// TIA Portal V20 export
// export: Created 2025-12-01T14:57:00.6413391Z, ExportSetting None, DisplayName Totally Integrated Automation Portal, DisplayVersion V20 Update 3, DisplayName TIA Portal Openness, DisplayVersion V20 Update 3, DisplayName TIA Portal Version Control Interface, DisplayVersion V20 Update 3, DisplayName STEP 7 Professional, DisplayVersion V20 Update 3, DisplayName STEP 7 Safety, DisplayVersion V20 Update 2, DisplayName WinCC Basic/Comfort/Advanced, DisplayVersion V20 Update 3, DisplayName WinCC Professional, DisplayVersion V20 Update 3, DisplayName WinCC Unified, DisplayVersion V20 Update 3
FUNCTION "FC452_TL_TR_E1E3_S2_Pres" : Void   // FC452, LAD
{ S7_Optimized_Access := 'FALSE' }
AUTHOR : TLigero
NAME : 20160208
VERSION : 3.1
// stored: AutoNumber false, SetENOAutomatically false
   VAR_INPUT
      Mesa : UInt;
      En_Tension : Bool;
      pHsMx_E1 : Bool;   // Para contar cuando se entra por E1
      pHsMx_E3 : Bool;   // Para contar cuando se entra por E3
      Termico_E1_Tx : Bool;
      Termico_S2_Tx : Bool;
      Avance_E1_Tx_Ok : Bool;
      Avance_E3_Tx_Ok : Bool;   // será el retroceso de E1
      Avance_S2_Tx_Ok : Bool;
      PosTR_E1 : Bool;
      PosTR_S2 : Bool;
      TP_E1E3_UP : Bool;
      TP_E1E3_DW : Bool;
      TP_E3E1_UP : Bool;
      TP_E3E1_DW : Bool;
      AVTF_Ent_M1 : Bool;
      AVTF_Ent_M3 : Bool;
      NXT_Avance : Bool;
      PTF_Mx_MSig : Bool;
      V_CNT_pHsMx_E1 : UDInt;
      V_CNT_pHsMx_E3 : UDInt;
      V_Paro : UDInt;
      V_CNT_ApHsMx : UDInt;
      V_TOut_Tx_Mx : UDInt;
      V_TOut_TR : UDInt;
      V_TOut_TP : UDInt;
      V_Reparto_E1_E3 : UDInt;
   END_VAR
   VAR_OUTPUT
      PTF_Ent_M1 : Bool;
      PTF_Ent_M3 : Bool;
      AVTF_Mx_MSig : Bool;
      NXT_Descarga_Act : Bool;
   END_VAR
   VAR_IN_OUT
      MemFP_Carga_E1 : Bool;
   END_VAR
   VAR_TEMP
      Mem_CNT_Aus : Bool;
      Aux_Parar : Bool;
      Mem_CNT_Pres : Bool;
      Mem_CNT_Tmp_Paro : Bool;
      TEMP_MA_TR_Pos_E1 : Bool;
      TEMP_MA_TR_Pos_S2 : Bool;
      Atasco : Bool;
      Tout_movimiento : Bool;
      tout_tope : Bool;
      ok_tension : Bool;
      V_Presencia : UDInt;
   END_VAR
   VAR_TEMP   // added for the SCL form of the ladder/FBD networks
      _w1 : Bool;
   END_VAR
BEGIN

REGION Network 1: Marca General Error
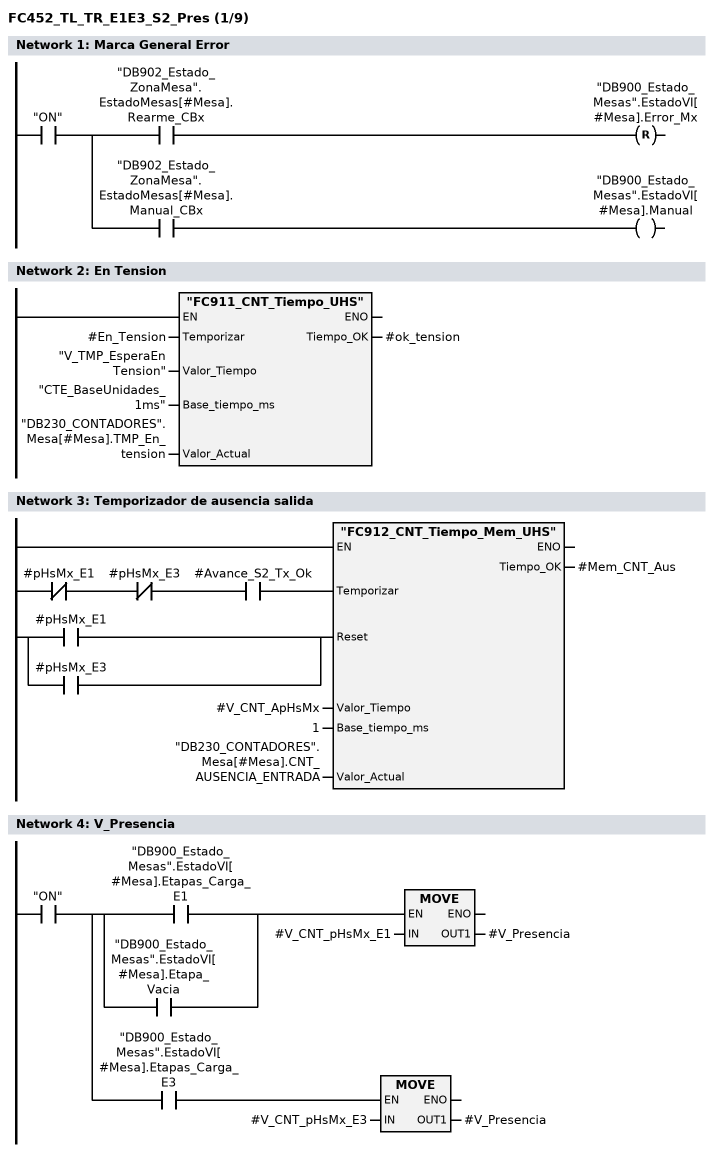
   RUNG wire#powerrail
      Contact( "ON" )
      wire#w1
      Contact( "DB902_Estado_ZonaMesa".EstadoMesas[#Mesa].Rearme_CBx )
      R_Coil( "DB900_Estado_Mesas".EstadoVI[#Mesa].Error_Mx )
   END_RUNG
   RUNG wire#w1
      Contact( "DB902_Estado_ZonaMesa".EstadoMesas[#Mesa].Manual_CBx )
      Coil( "DB900_Estado_Mesas".EstadoVI[#Mesa].Manual )
   END_RUNG
   // the same network as SCL:
   IF "ON" AND "DB902_Estado_ZonaMesa".EstadoMesas[#Mesa].Rearme_CBx THEN
       "DB900_Estado_Mesas".EstadoVI[#Mesa].Error_Mx := FALSE;
   END_IF;
   "DB900_Estado_Mesas".EstadoVI[#Mesa].Manual := "ON" AND "DB902_Estado_ZonaMesa".EstadoMesas[#Mesa].Manual_CBx;
END_REGION

REGION Network 2: En Tension
   RUNG wire#powerrail
      "FC911_CNT_Tiempo_UHS"(Temporizar := #En_Tension, Valor_Tiempo := "V_TMP_EsperaEnTension", Base_tiempo_ms := "CTE_BaseUnidades_1ms", Valor_Actual := "DB230_CONTADORES".Mesa[#Mesa].TMP_En_tension, Tiempo_OK => #ok_tension)
   END_RUNG
   // the same network as SCL:
   "FC911_CNT_Tiempo_UHS"(Temporizar := #En_Tension,
                          Valor_Tiempo := "V_TMP_EsperaEnTension",
                          Base_tiempo_ms := "CTE_BaseUnidades_1ms",
                          Valor_Actual := "DB230_CONTADORES".Mesa[#Mesa].TMP_En_tension,
                          Tiempo_OK => #ok_tension);
END_REGION

REGION Network 3: Temporizador de ausencia salida
   RUNG wire#powerrail
      "FC912_CNT_Tiempo_Mem_UHS"(Temporizar := wire#w1, Reset := wire#w2, Valor_Tiempo := #V_CNT_ApHsMx, Base_tiempo_ms := 1, Valor_Actual := "DB230_CONTADORES".Mesa[#Mesa].CNT_AUSENCIA_ENTRADA, Tiempo_OK => #Mem_CNT_Aus)
   END_RUNG
   RUNG wire#powerrail
      I_Contact( #pHsMx_E1 )
      I_Contact( #pHsMx_E3 )
      Contact( #Avance_S2_Tx_Ok )
   END_RUNG wire#w1
   RUNG wire#powerrail
      Contact( #pHsMx_E1 )
   END_RUNG wire#w2
   RUNG wire#powerrail
      Contact( #pHsMx_E3 )
   END_RUNG wire#w2
   // the same network as SCL:
   "FC912_CNT_Tiempo_Mem_UHS"(Temporizar := NOT #pHsMx_E1 AND NOT #pHsMx_E3 AND #Avance_S2_Tx_Ok,
                           Reset := #pHsMx_E1 OR #pHsMx_E3,
                           Valor_Tiempo := #V_CNT_ApHsMx,
                           Base_tiempo_ms := 1,
                           Valor_Actual := "DB230_CONTADORES".Mesa[#Mesa].CNT_AUSENCIA_ENTRADA,
                           Tiempo_OK => #Mem_CNT_Aus);
END_REGION

REGION Network 4: V_Presencia
   RUNG wire#powerrail
      Contact( "ON" )
      wire#w1
      Contact( "DB900_Estado_Mesas".EstadoVI[#Mesa].Etapas_Carga_E1 )
      wire#w2
      Move(in := #V_CNT_pHsMx_E1, out1 => #V_Presencia)
   END_RUNG
   RUNG wire#w1
      Contact( "DB900_Estado_Mesas".EstadoVI[#Mesa].Etapa_Vacia )
   END_RUNG wire#w2
   RUNG wire#w1
      Contact( "DB900_Estado_Mesas".EstadoVI[#Mesa].Etapas_Carga_E3 )
      Move(in := #V_CNT_pHsMx_E3, out1 => #V_Presencia)
   END_RUNG
   // the same network as SCL:
   IF "ON" AND ("DB900_Estado_Mesas".EstadoVI[#Mesa].Etapas_Carga_E1 OR "DB900_Estado_Mesas".EstadoVI[#Mesa].Etapa_Vacia) THEN
       #V_Presencia := #V_CNT_pHsMx_E1;
   END_IF;
   IF "ON" AND "DB900_Estado_Mesas".EstadoVI[#Mesa].Etapas_Carga_E3 THEN
       #V_Presencia := #V_CNT_pHsMx_E3;
   END_IF;
END_REGION

REGION Network 5: Temporizador presencia
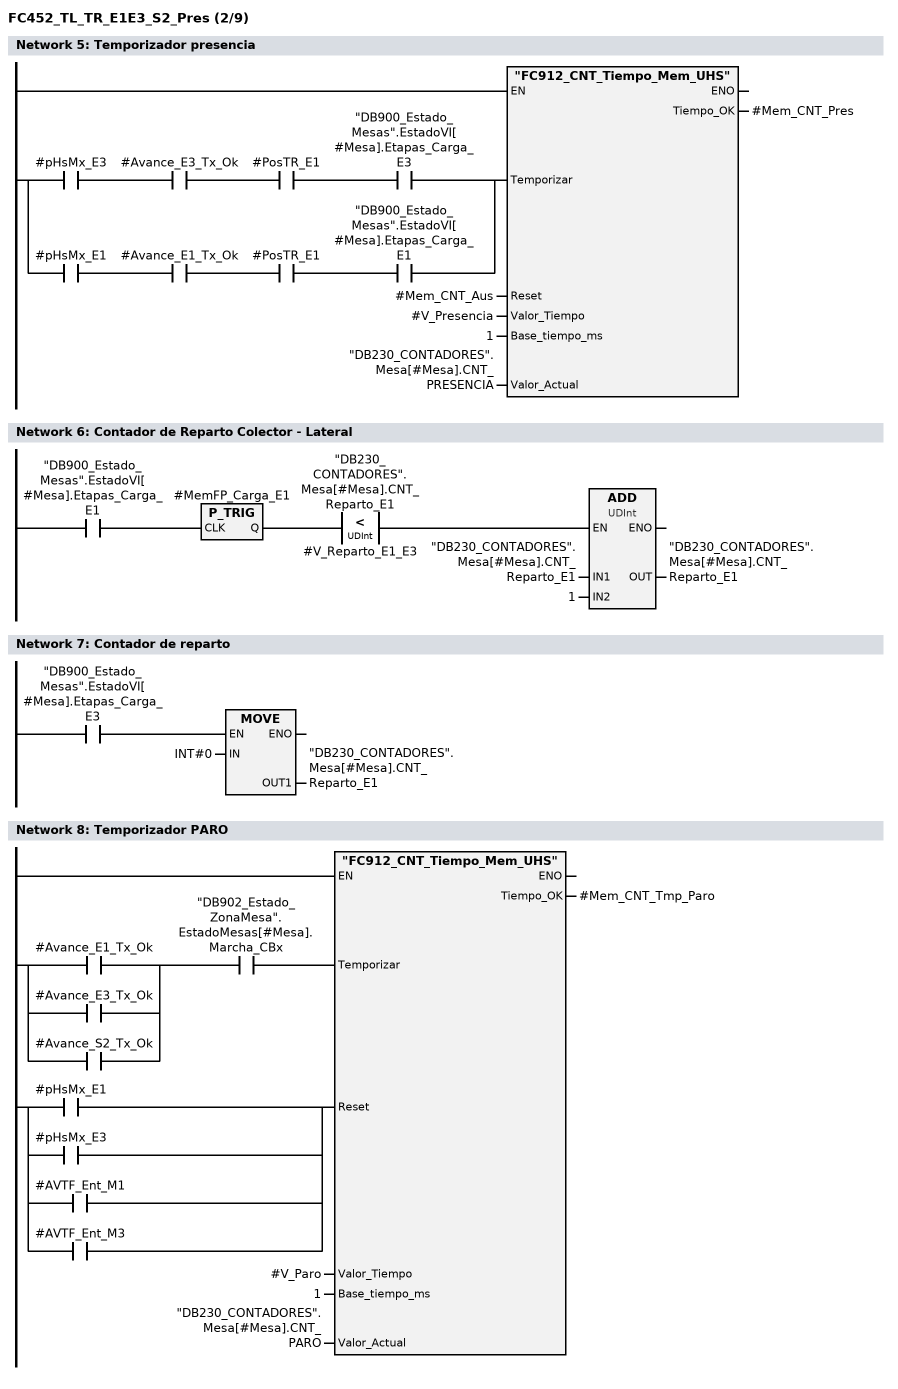
   RUNG wire#powerrail
      "FC912_CNT_Tiempo_Mem_UHS"(Temporizar := wire#w1, Reset := #Mem_CNT_Aus, Valor_Tiempo := #V_Presencia, Base_tiempo_ms := 1, Valor_Actual := "DB230_CONTADORES".Mesa[#Mesa].CNT_PRESENCIA, Tiempo_OK => #Mem_CNT_Pres)
   END_RUNG
   RUNG wire#powerrail
      Contact( #pHsMx_E3 )
      Contact( #Avance_E3_Tx_Ok )
      Contact( #PosTR_E1 )
      Contact( "DB900_Estado_Mesas".EstadoVI[#Mesa].Etapas_Carga_E3 )
   END_RUNG wire#w1
   RUNG wire#powerrail
      Contact( #pHsMx_E1 )
      Contact( #Avance_E1_Tx_Ok )
      Contact( #PosTR_E1 )
      Contact( "DB900_Estado_Mesas".EstadoVI[#Mesa].Etapas_Carga_E1 )
   END_RUNG wire#w1
   // the same network as SCL:
   "FC912_CNT_Tiempo_Mem_UHS"(Temporizar := (#pHsMx_E3 AND #Avance_E3_Tx_Ok AND #PosTR_E1 AND "DB900_Estado_Mesas".EstadoVI[#Mesa].Etapas_Carga_E3) OR (#pHsMx_E1 AND #Avance_E1_Tx_Ok AND #PosTR_E1 AND "DB900_Estado_Mesas".EstadoVI[#Mesa].Etapas_Carga_E1),
                           Reset := #Mem_CNT_Aus,
                           Valor_Tiempo := #V_Presencia,
                           Base_tiempo_ms := 1,
                           Valor_Actual := "DB230_CONTADORES".Mesa[#Mesa].CNT_PRESENCIA,
                           Tiempo_OK => #Mem_CNT_Pres);
END_REGION

REGION Network 6: Contador de Reparto Colector - Lateral
   RUNG wire#powerrail
      Contact( "DB900_Estado_Mesas".EstadoVI[#Mesa].Etapas_Carga_E1 )
      P_Trig( #MemFP_Carga_E1 )
      { S7_Templates := "SrcType := UDInt" } LT_Contact(in1 := "DB230_CONTADORES".Mesa[#Mesa].CNT_Reparto_E1, in2 := #V_Reparto_E1_E3)
      { S7_Templates := "SrcType := UDInt"; S7_GenerateENO := "TRUE" } Add(in1 := "DB230_CONTADORES".Mesa[#Mesa].CNT_Reparto_E1, in2 := 1, out => "DB230_CONTADORES".Mesa[#Mesa].CNT_Reparto_E1)
   END_RUNG
   // the same network as SCL:
   #_w1 := "DB900_Estado_Mesas".EstadoVI[#Mesa].Etapas_Carga_E1 AND NOT #MemFP_Carga_E1;   // rising edge
   #MemFP_Carga_E1 := "DB900_Estado_Mesas".EstadoVI[#Mesa].Etapas_Carga_E1;
   IF #_w1 AND ("DB230_CONTADORES".Mesa[#Mesa].CNT_Reparto_E1 < #V_Reparto_E1_E3) THEN
       "DB230_CONTADORES".Mesa[#Mesa].CNT_Reparto_E1 := "DB230_CONTADORES".Mesa[#Mesa].CNT_Reparto_E1 + 1;
   END_IF;
END_REGION

REGION Network 7: Contador de reparto
   RUNG wire#powerrail
      Contact( "DB900_Estado_Mesas".EstadoVI[#Mesa].Etapas_Carga_E3 )
      { S7_GenerateENO := "TRUE" } Move(in := INT#0, out1 => "DB230_CONTADORES".Mesa[#Mesa].CNT_Reparto_E1)
   END_RUNG
   // the same network as SCL:
   IF "DB900_Estado_Mesas".EstadoVI[#Mesa].Etapas_Carga_E3 THEN
       "DB230_CONTADORES".Mesa[#Mesa].CNT_Reparto_E1 := INT#0;
   END_IF;
END_REGION

REGION Network 8: Temporizador PARO
   RUNG wire#powerrail
      "FC912_CNT_Tiempo_Mem_UHS"(Temporizar := wire#w2, Reset := wire#w3, Valor_Tiempo := #V_Paro, Base_tiempo_ms := 1, Valor_Actual := "DB230_CONTADORES".Mesa[#Mesa].CNT_PARO, Tiempo_OK => #Mem_CNT_Tmp_Paro)
   END_RUNG
   RUNG wire#powerrail
      Contact( #Avance_E1_Tx_Ok )
      wire#w1
      Contact( "DB902_Estado_ZonaMesa".EstadoMesas[#Mesa].Marcha_CBx )
   END_RUNG wire#w2
   RUNG wire#powerrail
      Contact( #Avance_E3_Tx_Ok )
   END_RUNG wire#w1
   RUNG wire#powerrail
      Contact( #Avance_S2_Tx_Ok )
   END_RUNG wire#w1
   RUNG wire#powerrail
      Contact( #pHsMx_E1 )
   END_RUNG wire#w3
   RUNG wire#powerrail
      Contact( #pHsMx_E3 )
   END_RUNG wire#w3
   RUNG wire#powerrail
      Contact( #AVTF_Ent_M1 )
   END_RUNG wire#w3
   RUNG wire#powerrail
      Contact( #AVTF_Ent_M3 )
   END_RUNG wire#w3
   // the same network as SCL:
   "FC912_CNT_Tiempo_Mem_UHS"(Temporizar := (#Avance_E1_Tx_Ok OR #Avance_E3_Tx_Ok OR #Avance_S2_Tx_Ok) AND "DB902_Estado_ZonaMesa".EstadoMesas[#Mesa].Marcha_CBx,
                           Reset := #pHsMx_E1 OR #pHsMx_E3 OR #AVTF_Ent_M1 OR #AVTF_Ent_M3,
                           Valor_Tiempo := #V_Paro,
                           Base_tiempo_ms := 1,
                           Valor_Actual := "DB230_CONTADORES".Mesa[#Mesa].CNT_PARO,
                           Tiempo_OK => #Mem_CNT_Tmp_Paro);
END_REGION

REGION Network 9: Etapas_Carga_E1
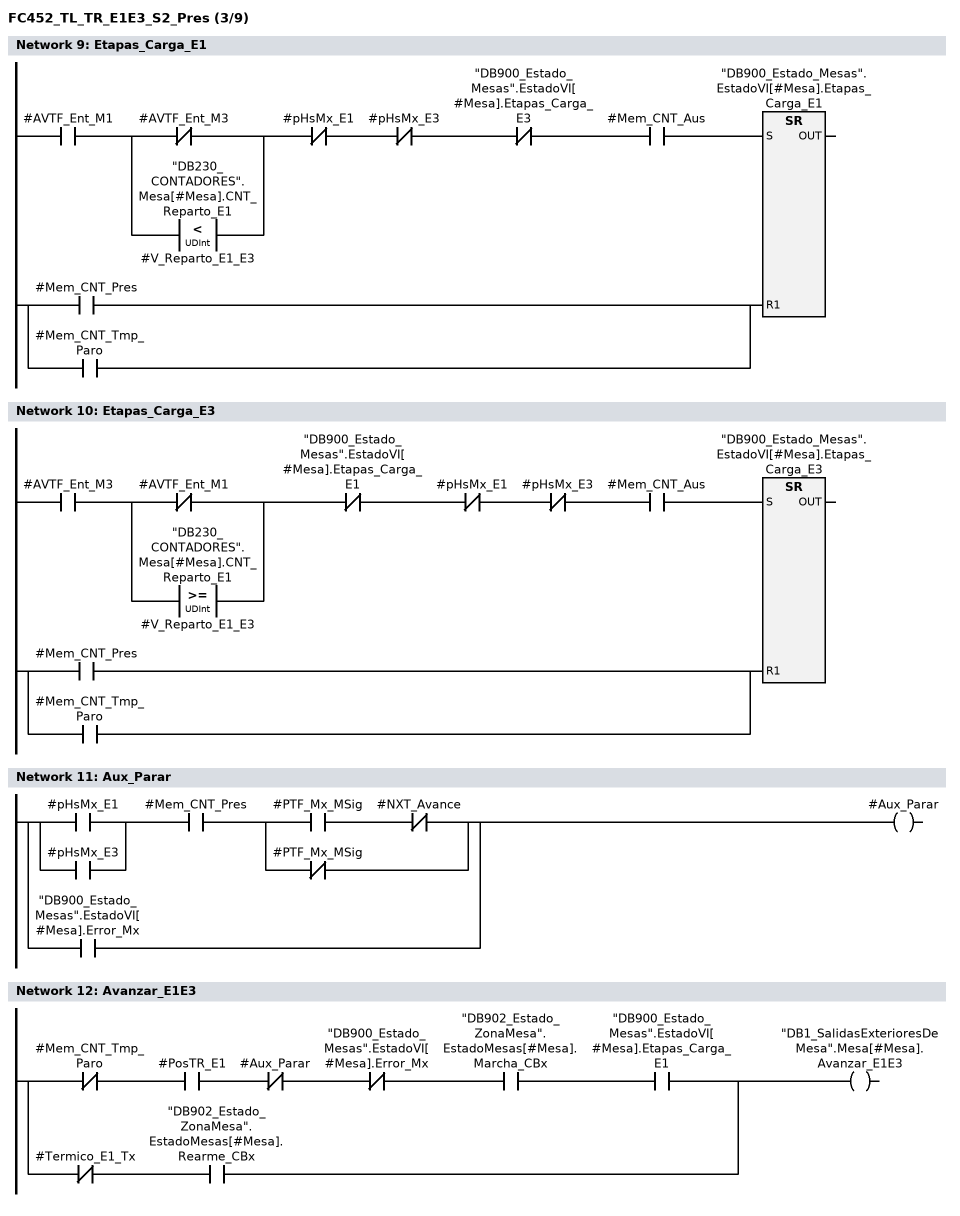
   RUNG wire#powerrail
      Contact( #AVTF_Ent_M1 )
      wire#w1
      I_Contact( #AVTF_Ent_M3 )
      wire#w2
      I_Contact( #pHsMx_E1 )
      I_Contact( #pHsMx_E3 )
      I_Contact( "DB900_Estado_Mesas".EstadoVI[#Mesa].Etapas_Carga_E3 )
      Contact( #Mem_CNT_Aus )
      S_SR(operand := "DB900_Estado_Mesas".EstadoVI[#Mesa].Etapas_Carga_E1, r1 := wire#w3)
   END_RUNG
   RUNG wire#w1
      { S7_Templates := "SrcType := UDInt" } LT_Contact(in1 := "DB230_CONTADORES".Mesa[#Mesa].CNT_Reparto_E1, in2 := #V_Reparto_E1_E3)
   END_RUNG wire#w2
   RUNG wire#powerrail
      Contact( #Mem_CNT_Pres )
   END_RUNG wire#w3
   RUNG wire#powerrail
      Contact( #Mem_CNT_Tmp_Paro )
   END_RUNG wire#w3
   // the same network as SCL:
   IF #AVTF_Ent_M1 AND (NOT #AVTF_Ent_M3 OR ("DB230_CONTADORES".Mesa[#Mesa].CNT_Reparto_E1 < #V_Reparto_E1_E3)) AND NOT #pHsMx_E1 AND NOT #pHsMx_E3 AND NOT "DB900_Estado_Mesas".EstadoVI[#Mesa].Etapas_Carga_E3 AND #Mem_CNT_Aus THEN
       "DB900_Estado_Mesas".EstadoVI[#Mesa].Etapas_Carga_E1 := TRUE;   // SR flip-flop
   END_IF;
   IF #Mem_CNT_Pres OR #Mem_CNT_Tmp_Paro THEN
       "DB900_Estado_Mesas".EstadoVI[#Mesa].Etapas_Carga_E1 := FALSE;
   END_IF;
END_REGION

REGION Network 10: Etapas_Carga_E3
   RUNG wire#powerrail
      Contact( #AVTF_Ent_M3 )
      wire#w1
      I_Contact( #AVTF_Ent_M1 )
      wire#w2
      I_Contact( "DB900_Estado_Mesas".EstadoVI[#Mesa].Etapas_Carga_E1 )
      I_Contact( #pHsMx_E1 )
      I_Contact( #pHsMx_E3 )
      Contact( #Mem_CNT_Aus )
      S_SR(operand := "DB900_Estado_Mesas".EstadoVI[#Mesa].Etapas_Carga_E3, r1 := wire#w3)
   END_RUNG
   RUNG wire#w1
      { S7_Templates := "SrcType := UDInt" } GE_Contact(in1 := "DB230_CONTADORES".Mesa[#Mesa].CNT_Reparto_E1, in2 := #V_Reparto_E1_E3)
   END_RUNG wire#w2
   RUNG wire#powerrail
      Contact( #Mem_CNT_Pres )
   END_RUNG wire#w3
   RUNG wire#powerrail
      Contact( #Mem_CNT_Tmp_Paro )
   END_RUNG wire#w3
   // the same network as SCL:
   IF #AVTF_Ent_M3 AND (NOT #AVTF_Ent_M1 OR ("DB230_CONTADORES".Mesa[#Mesa].CNT_Reparto_E1 >= #V_Reparto_E1_E3)) AND NOT "DB900_Estado_Mesas".EstadoVI[#Mesa].Etapas_Carga_E1 AND NOT #pHsMx_E1 AND NOT #pHsMx_E3 AND #Mem_CNT_Aus THEN
       "DB900_Estado_Mesas".EstadoVI[#Mesa].Etapas_Carga_E3 := TRUE;   // SR flip-flop
   END_IF;
   IF #Mem_CNT_Pres OR #Mem_CNT_Tmp_Paro THEN
       "DB900_Estado_Mesas".EstadoVI[#Mesa].Etapas_Carga_E3 := FALSE;
   END_IF;
END_REGION

REGION Network 11: Aux_Parar
   RUNG wire#powerrail
      Contact( #pHsMx_E1 )
      wire#w1
      Contact( #Mem_CNT_Pres )
      wire#w2
      Contact( #PTF_Mx_MSig )
      I_Contact( #NXT_Avance )
      wire#w3
      Coil( #Aux_Parar )
   END_RUNG
   RUNG wire#powerrail
      Contact( #pHsMx_E3 )
   END_RUNG wire#w1
   RUNG wire#w2
      I_Contact( #PTF_Mx_MSig )
   END_RUNG wire#w3
   RUNG wire#powerrail
      Contact( "DB900_Estado_Mesas".EstadoVI[#Mesa].Error_Mx )
   END_RUNG wire#w3
   // the same network as SCL:
   #Aux_Parar := ((#pHsMx_E1 OR #pHsMx_E3) AND #Mem_CNT_Pres AND ((#PTF_Mx_MSig AND NOT #NXT_Avance) OR NOT #PTF_Mx_MSig)) OR "DB900_Estado_Mesas".EstadoVI[#Mesa].Error_Mx;
END_REGION

REGION Network 12: Avanzar_E1E3
   RUNG wire#powerrail
      I_Contact( #Mem_CNT_Tmp_Paro )
      Contact( #PosTR_E1 )
      I_Contact( #Aux_Parar )
      I_Contact( "DB900_Estado_Mesas".EstadoVI[#Mesa].Error_Mx )
      Contact( "DB902_Estado_ZonaMesa".EstadoMesas[#Mesa].Marcha_CBx )
      Contact( "DB900_Estado_Mesas".EstadoVI[#Mesa].Etapas_Carga_E1 )
      wire#w1
      Coil( "DB1_SalidasExterioresDeMesa".Mesa[#Mesa].Avanzar_E1E3 )
   END_RUNG
   RUNG wire#powerrail
      I_Contact( #Termico_E1_Tx )
      Contact( "DB902_Estado_ZonaMesa".EstadoMesas[#Mesa].Rearme_CBx )
   END_RUNG wire#w1
   // the same network as SCL:
   "DB1_SalidasExterioresDeMesa".Mesa[#Mesa].Avanzar_E1E3 := (NOT #Mem_CNT_Tmp_Paro AND #PosTR_E1 AND NOT #Aux_Parar AND NOT "DB900_Estado_Mesas".EstadoVI[#Mesa].Error_Mx AND "DB902_Estado_ZonaMesa".EstadoMesas[#Mesa].Marcha_CBx AND "DB900_Estado_Mesas".EstadoVI[#Mesa].Etapas_Carga_E1) OR (NOT #Termico_E1_Tx AND "DB902_Estado_ZonaMesa".EstadoMesas[#Mesa].Rearme_CBx);
END_REGION

REGION Network 13: Retroceder_E1E3
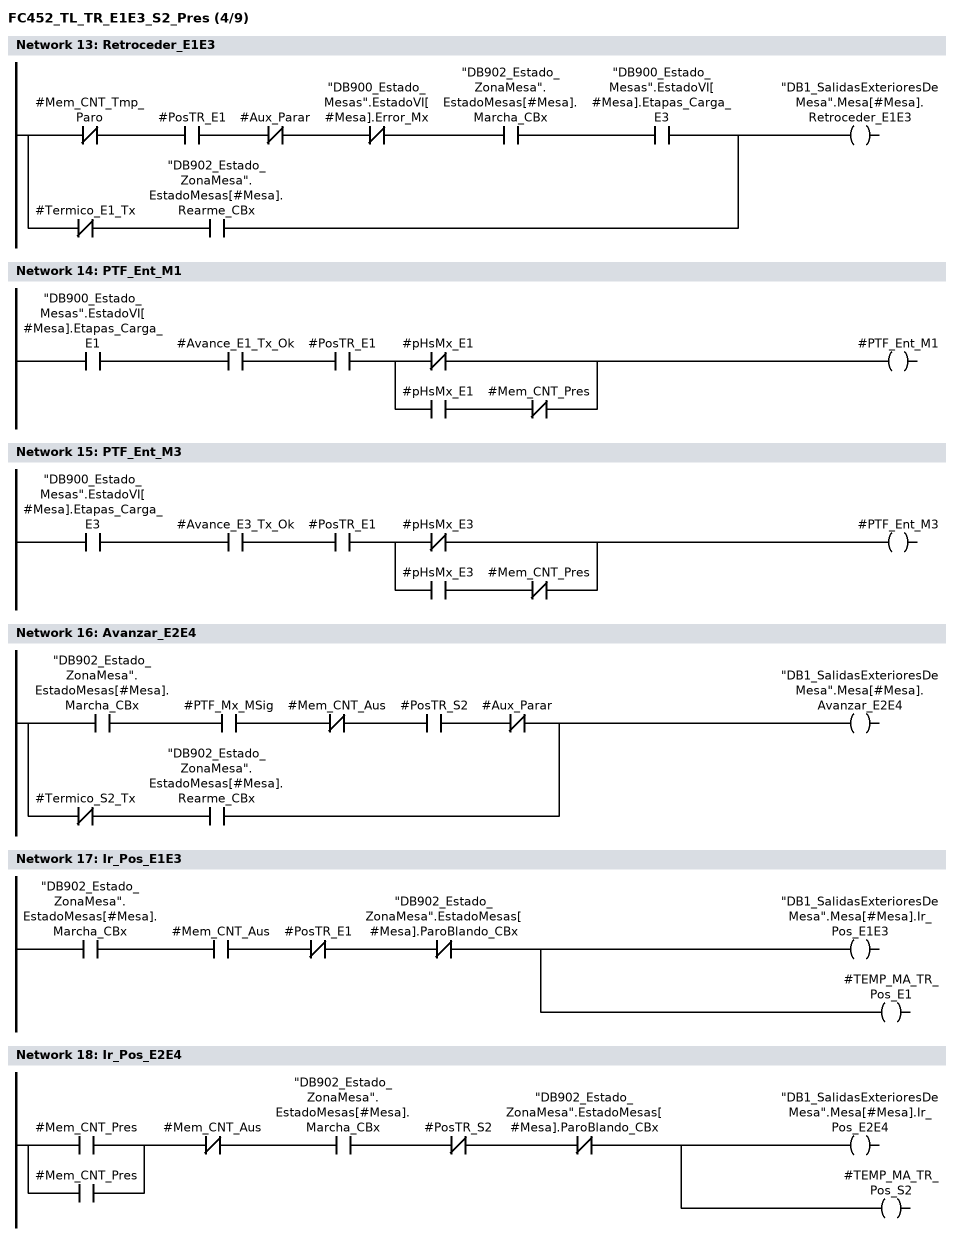
   RUNG wire#powerrail
      I_Contact( #Mem_CNT_Tmp_Paro )
      Contact( #PosTR_E1 )
      I_Contact( #Aux_Parar )
      I_Contact( "DB900_Estado_Mesas".EstadoVI[#Mesa].Error_Mx )
      Contact( "DB902_Estado_ZonaMesa".EstadoMesas[#Mesa].Marcha_CBx )
      Contact( "DB900_Estado_Mesas".EstadoVI[#Mesa].Etapas_Carga_E3 )
      wire#w1
      Coil( "DB1_SalidasExterioresDeMesa".Mesa[#Mesa].Retroceder_E1E3 )
   END_RUNG
   RUNG wire#powerrail
      I_Contact( #Termico_E1_Tx )
      Contact( "DB902_Estado_ZonaMesa".EstadoMesas[#Mesa].Rearme_CBx )
   END_RUNG wire#w1
   // the same network as SCL:
   "DB1_SalidasExterioresDeMesa".Mesa[#Mesa].Retroceder_E1E3 := (NOT #Mem_CNT_Tmp_Paro AND #PosTR_E1 AND NOT #Aux_Parar AND NOT "DB900_Estado_Mesas".EstadoVI[#Mesa].Error_Mx AND "DB902_Estado_ZonaMesa".EstadoMesas[#Mesa].Marcha_CBx AND "DB900_Estado_Mesas".EstadoVI[#Mesa].Etapas_Carga_E3) OR (NOT #Termico_E1_Tx AND "DB902_Estado_ZonaMesa".EstadoMesas[#Mesa].Rearme_CBx);
END_REGION

REGION Network 14: PTF_Ent_M1
   RUNG wire#powerrail
      Contact( "DB900_Estado_Mesas".EstadoVI[#Mesa].Etapas_Carga_E1 )
      Contact( #Avance_E1_Tx_Ok )
      Contact( #PosTR_E1 )
      wire#w1
      I_Contact( #pHsMx_E1 )
      wire#w2
      Coil( #PTF_Ent_M1 )
   END_RUNG
   RUNG wire#w1
      Contact( #pHsMx_E1 )
      I_Contact( #Mem_CNT_Pres )
   END_RUNG wire#w2
   // the same network as SCL:
   #PTF_Ent_M1 := "DB900_Estado_Mesas".EstadoVI[#Mesa].Etapas_Carga_E1 AND #Avance_E1_Tx_Ok AND #PosTR_E1 AND (NOT #pHsMx_E1 OR (#pHsMx_E1 AND NOT #Mem_CNT_Pres));
END_REGION

REGION Network 15: PTF_Ent_M3
   RUNG wire#powerrail
      Contact( "DB900_Estado_Mesas".EstadoVI[#Mesa].Etapas_Carga_E3 )
      Contact( #Avance_E3_Tx_Ok )
      Contact( #PosTR_E1 )
      wire#w1
      I_Contact( #pHsMx_E3 )
      wire#w2
      Coil( #PTF_Ent_M3 )
   END_RUNG
   RUNG wire#w1
      Contact( #pHsMx_E3 )
      I_Contact( #Mem_CNT_Pres )
   END_RUNG wire#w2
   // the same network as SCL:
   #PTF_Ent_M3 := "DB900_Estado_Mesas".EstadoVI[#Mesa].Etapas_Carga_E3 AND #Avance_E3_Tx_Ok AND #PosTR_E1 AND (NOT #pHsMx_E3 OR (#pHsMx_E3 AND NOT #Mem_CNT_Pres));
END_REGION

REGION Network 16: Avanzar_E2E4
   RUNG wire#powerrail
      Contact( "DB902_Estado_ZonaMesa".EstadoMesas[#Mesa].Marcha_CBx )
      Contact( #PTF_Mx_MSig )
      I_Contact( #Mem_CNT_Aus )
      Contact( #PosTR_S2 )
      I_Contact( #Aux_Parar )
      wire#w1
      Coil( "DB1_SalidasExterioresDeMesa".Mesa[#Mesa].Avanzar_E2E4 )
   END_RUNG
   RUNG wire#powerrail
      I_Contact( #Termico_S2_Tx )
      Contact( "DB902_Estado_ZonaMesa".EstadoMesas[#Mesa].Rearme_CBx )
   END_RUNG wire#w1
   // the same network as SCL:
   "DB1_SalidasExterioresDeMesa".Mesa[#Mesa].Avanzar_E2E4 := ("DB902_Estado_ZonaMesa".EstadoMesas[#Mesa].Marcha_CBx AND #PTF_Mx_MSig AND NOT #Mem_CNT_Aus AND #PosTR_S2 AND NOT #Aux_Parar) OR (NOT #Termico_S2_Tx AND "DB902_Estado_ZonaMesa".EstadoMesas[#Mesa].Rearme_CBx);
END_REGION

REGION Network 17: Ir_Pos_E1E3
   RUNG wire#powerrail
      Contact( "DB902_Estado_ZonaMesa".EstadoMesas[#Mesa].Marcha_CBx )
      Contact( #Mem_CNT_Aus )
      I_Contact( #PosTR_E1 )
      I_Contact( "DB902_Estado_ZonaMesa".EstadoMesas[#Mesa].ParoBlando_CBx )
      wire#w1
      Coil( "DB1_SalidasExterioresDeMesa".Mesa[#Mesa].Ir_Pos_E1E3 )
   END_RUNG
   RUNG wire#w1
      Coil( #TEMP_MA_TR_Pos_E1 )
   END_RUNG
   // the same network as SCL:
   #_w1 := "DB902_Estado_ZonaMesa".EstadoMesas[#Mesa].Marcha_CBx AND #Mem_CNT_Aus AND NOT #PosTR_E1 AND NOT "DB902_Estado_ZonaMesa".EstadoMesas[#Mesa].ParoBlando_CBx;
   "DB1_SalidasExterioresDeMesa".Mesa[#Mesa].Ir_Pos_E1E3 := "DB902_Estado_ZonaMesa".EstadoMesas[#Mesa].Marcha_CBx AND #Mem_CNT_Aus AND NOT #PosTR_E1 AND NOT "DB902_Estado_ZonaMesa".EstadoMesas[#Mesa].ParoBlando_CBx;
   #TEMP_MA_TR_Pos_E1 := #_w1;
END_REGION

REGION Network 18: Ir_Pos_E2E4
   RUNG wire#powerrail
      Contact( #Mem_CNT_Pres )
      wire#w1
      I_Contact( #Mem_CNT_Aus )
      Contact( "DB902_Estado_ZonaMesa".EstadoMesas[#Mesa].Marcha_CBx )
      I_Contact( #PosTR_S2 )
      I_Contact( "DB902_Estado_ZonaMesa".EstadoMesas[#Mesa].ParoBlando_CBx )
      wire#w2
      Coil( "DB1_SalidasExterioresDeMesa".Mesa[#Mesa].Ir_Pos_E2E4 )
   END_RUNG
   RUNG wire#powerrail
      Contact( #Mem_CNT_Pres )
   END_RUNG wire#w1
   RUNG wire#w2
      Coil( #TEMP_MA_TR_Pos_S2 )
   END_RUNG
   // the same network as SCL:
   #_w1 := (#Mem_CNT_Pres OR #Mem_CNT_Pres) AND NOT #Mem_CNT_Aus AND "DB902_Estado_ZonaMesa".EstadoMesas[#Mesa].Marcha_CBx AND NOT #PosTR_S2 AND NOT "DB902_Estado_ZonaMesa".EstadoMesas[#Mesa].ParoBlando_CBx;
   "DB1_SalidasExterioresDeMesa".Mesa[#Mesa].Ir_Pos_E2E4 := (#Mem_CNT_Pres OR #Mem_CNT_Pres) AND NOT #Mem_CNT_Aus AND "DB902_Estado_ZonaMesa".EstadoMesas[#Mesa].Marcha_CBx AND NOT #PosTR_S2 AND NOT "DB902_Estado_ZonaMesa".EstadoMesas[#Mesa].ParoBlando_CBx;
   #TEMP_MA_TR_Pos_S2 := #_w1;
END_REGION

REGION Network 19: Subir Topes
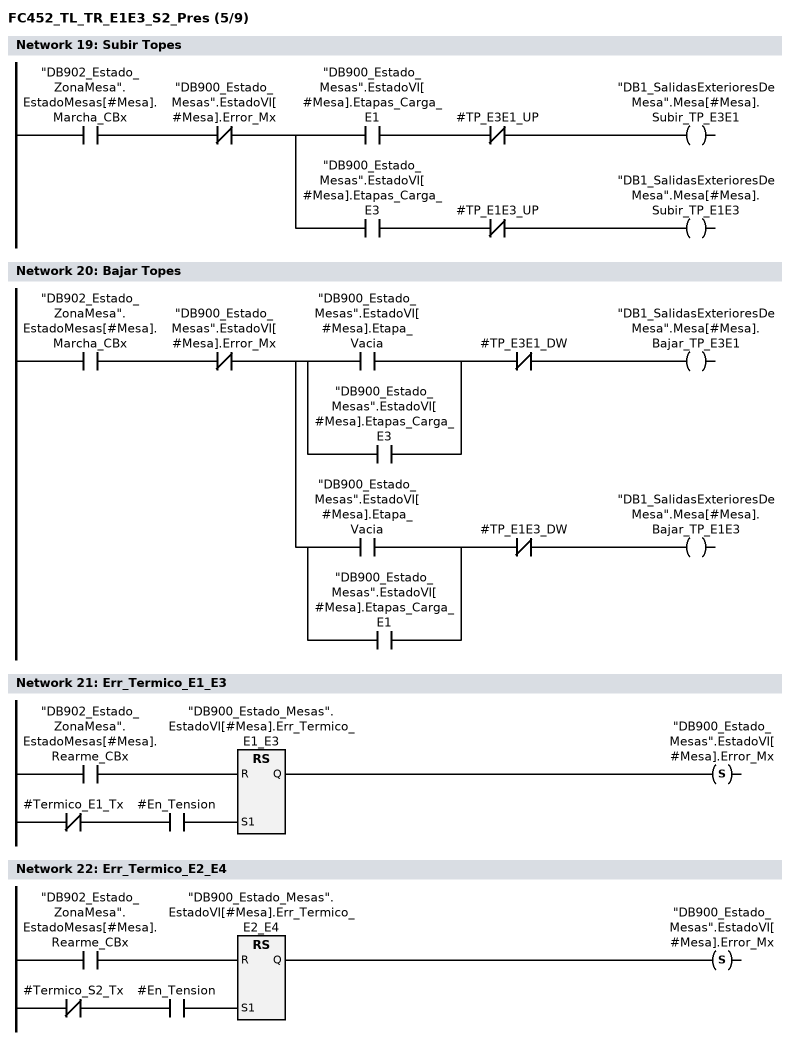
   RUNG wire#powerrail
      Contact( "DB902_Estado_ZonaMesa".EstadoMesas[#Mesa].Marcha_CBx )
      I_Contact( "DB900_Estado_Mesas".EstadoVI[#Mesa].Error_Mx )
      wire#w1
      Contact( "DB900_Estado_Mesas".EstadoVI[#Mesa].Etapas_Carga_E1 )
      I_Contact( #TP_E3E1_UP )
      Coil( "DB1_SalidasExterioresDeMesa".Mesa[#Mesa].Subir_TP_E3E1 )
   END_RUNG
   RUNG wire#w1
      Contact( "DB900_Estado_Mesas".EstadoVI[#Mesa].Etapas_Carga_E3 )
      I_Contact( #TP_E1E3_UP )
      Coil( "DB1_SalidasExterioresDeMesa".Mesa[#Mesa].Subir_TP_E1E3 )
   END_RUNG
   // the same network as SCL:
   #_w1 := "DB902_Estado_ZonaMesa".EstadoMesas[#Mesa].Marcha_CBx AND NOT "DB900_Estado_Mesas".EstadoVI[#Mesa].Error_Mx;
   "DB1_SalidasExterioresDeMesa".Mesa[#Mesa].Subir_TP_E3E1 := #_w1 AND "DB900_Estado_Mesas".EstadoVI[#Mesa].Etapas_Carga_E1 AND NOT #TP_E3E1_UP;
   "DB1_SalidasExterioresDeMesa".Mesa[#Mesa].Subir_TP_E1E3 := #_w1 AND "DB900_Estado_Mesas".EstadoVI[#Mesa].Etapas_Carga_E3 AND NOT #TP_E1E3_UP;
END_REGION

REGION Network 20: Bajar Topes
   RUNG wire#powerrail
      Contact( "DB902_Estado_ZonaMesa".EstadoMesas[#Mesa].Marcha_CBx )
      I_Contact( "DB900_Estado_Mesas".EstadoVI[#Mesa].Error_Mx )
      wire#w1
      Contact( "DB900_Estado_Mesas".EstadoVI[#Mesa].Etapa_Vacia )
      wire#w2
      I_Contact( #TP_E3E1_DW )
      Coil( "DB1_SalidasExterioresDeMesa".Mesa[#Mesa].Bajar_TP_E3E1 )
   END_RUNG
   RUNG wire#w1
      Contact( "DB900_Estado_Mesas".EstadoVI[#Mesa].Etapas_Carga_E3 )
   END_RUNG wire#w2
   RUNG wire#w1
      Contact( "DB900_Estado_Mesas".EstadoVI[#Mesa].Etapa_Vacia )
      wire#w3
      I_Contact( #TP_E1E3_DW )
      Coil( "DB1_SalidasExterioresDeMesa".Mesa[#Mesa].Bajar_TP_E1E3 )
   END_RUNG
   RUNG wire#w1
      Contact( "DB900_Estado_Mesas".EstadoVI[#Mesa].Etapas_Carga_E1 )
   END_RUNG wire#w3
   // the same network as SCL:
   #_w1 := "DB902_Estado_ZonaMesa".EstadoMesas[#Mesa].Marcha_CBx AND NOT "DB900_Estado_Mesas".EstadoVI[#Mesa].Error_Mx;
   "DB1_SalidasExterioresDeMesa".Mesa[#Mesa].Bajar_TP_E3E1 := #_w1 AND ("DB900_Estado_Mesas".EstadoVI[#Mesa].Etapa_Vacia OR "DB900_Estado_Mesas".EstadoVI[#Mesa].Etapas_Carga_E3) AND NOT #TP_E3E1_DW;
   "DB1_SalidasExterioresDeMesa".Mesa[#Mesa].Bajar_TP_E1E3 := #_w1 AND ("DB900_Estado_Mesas".EstadoVI[#Mesa].Etapa_Vacia OR "DB900_Estado_Mesas".EstadoVI[#Mesa].Etapas_Carga_E1) AND NOT #TP_E1E3_DW;
END_REGION

REGION Network 21: Err_Termico_E1_E3
   RUNG wire#powerrail
      Contact( "DB902_Estado_ZonaMesa".EstadoMesas[#Mesa].Rearme_CBx )
      S_RS(operand := "DB900_Estado_Mesas".EstadoVI[#Mesa].Err_Termico_E1_E3, s1 := wire#w1)
      S_Coil( "DB900_Estado_Mesas".EstadoVI[#Mesa].Error_Mx )
   END_RUNG
   RUNG wire#powerrail
      I_Contact( #Termico_E1_Tx )
      Contact( #En_Tension )
   END_RUNG wire#w1
   // the same network as SCL:
   IF "DB902_Estado_ZonaMesa".EstadoMesas[#Mesa].Rearme_CBx THEN
       "DB900_Estado_Mesas".EstadoVI[#Mesa].Err_Termico_E1_E3 := FALSE;   // RS flip-flop
   END_IF;
   IF NOT #Termico_E1_Tx AND #En_Tension THEN
       "DB900_Estado_Mesas".EstadoVI[#Mesa].Err_Termico_E1_E3 := TRUE;
   END_IF;
   IF "DB900_Estado_Mesas".EstadoVI[#Mesa].Err_Termico_E1_E3 THEN
       "DB900_Estado_Mesas".EstadoVI[#Mesa].Error_Mx := TRUE;
   END_IF;
END_REGION

REGION Network 22: Err_Termico_E2_E4
   RUNG wire#powerrail
      Contact( "DB902_Estado_ZonaMesa".EstadoMesas[#Mesa].Rearme_CBx )
      S_RS(operand := "DB900_Estado_Mesas".EstadoVI[#Mesa].Err_Termico_E2_E4, s1 := wire#w1)
      S_Coil( "DB900_Estado_Mesas".EstadoVI[#Mesa].Error_Mx )
   END_RUNG
   RUNG wire#powerrail
      I_Contact( #Termico_S2_Tx )
      Contact( #En_Tension )
   END_RUNG wire#w1
   // the same network as SCL:
   IF "DB902_Estado_ZonaMesa".EstadoMesas[#Mesa].Rearme_CBx THEN
       "DB900_Estado_Mesas".EstadoVI[#Mesa].Err_Termico_E2_E4 := FALSE;   // RS flip-flop
   END_IF;
   IF NOT #Termico_S2_Tx AND #En_Tension THEN
       "DB900_Estado_Mesas".EstadoVI[#Mesa].Err_Termico_E2_E4 := TRUE;
   END_IF;
   IF "DB900_Estado_Mesas".EstadoVI[#Mesa].Err_Termico_E2_E4 THEN
       "DB900_Estado_Mesas".EstadoVI[#Mesa].Error_Mx := TRUE;
   END_IF;
END_REGION

REGION Network 23: timeout movimiento tope
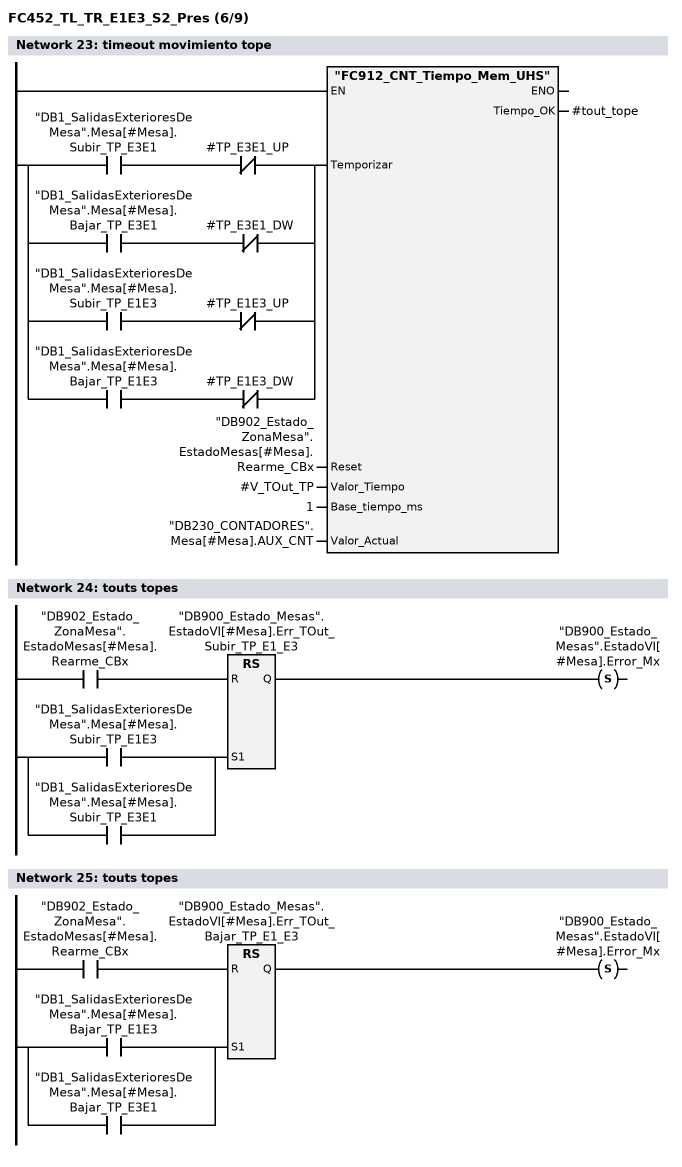
   RUNG wire#powerrail
      "FC912_CNT_Tiempo_Mem_UHS"(Temporizar := wire#w1, Reset := "DB902_Estado_ZonaMesa".EstadoMesas[#Mesa].Rearme_CBx, Valor_Tiempo := #V_TOut_TP, Base_tiempo_ms := 1, Valor_Actual := "DB230_CONTADORES".Mesa[#Mesa].AUX_CNT, Tiempo_OK => #tout_tope)
   END_RUNG
   RUNG wire#powerrail
      Contact( "DB1_SalidasExterioresDeMesa".Mesa[#Mesa].Subir_TP_E3E1 )
      I_Contact( #TP_E3E1_UP )
   END_RUNG wire#w1
   RUNG wire#powerrail
      Contact( "DB1_SalidasExterioresDeMesa".Mesa[#Mesa].Bajar_TP_E3E1 )
      I_Contact( #TP_E3E1_DW )
   END_RUNG wire#w1
   RUNG wire#powerrail
      Contact( "DB1_SalidasExterioresDeMesa".Mesa[#Mesa].Subir_TP_E1E3 )
      I_Contact( #TP_E1E3_UP )
   END_RUNG wire#w1
   RUNG wire#powerrail
      Contact( "DB1_SalidasExterioresDeMesa".Mesa[#Mesa].Bajar_TP_E1E3 )
      I_Contact( #TP_E1E3_DW )
   END_RUNG wire#w1
   // the same network as SCL:
   "FC912_CNT_Tiempo_Mem_UHS"(Temporizar := ("DB1_SalidasExterioresDeMesa".Mesa[#Mesa].Subir_TP_E3E1 AND NOT #TP_E3E1_UP) OR ("DB1_SalidasExterioresDeMesa".Mesa[#Mesa].Bajar_TP_E3E1 AND NOT #TP_E3E1_DW) OR ("DB1_SalidasExterioresDeMesa".Mesa[#Mesa].Subir_TP_E1E3 AND NOT #TP_E1E3_UP) OR ("DB1_SalidasExterioresDeMesa".Mesa[#Mesa].Bajar_TP_E1E3 AND NOT #TP_E1E3_DW),
                           Reset := "DB902_Estado_ZonaMesa".EstadoMesas[#Mesa].Rearme_CBx,
                           Valor_Tiempo := #V_TOut_TP,
                           Base_tiempo_ms := 1,
                           Valor_Actual := "DB230_CONTADORES".Mesa[#Mesa].AUX_CNT,
                           Tiempo_OK => #tout_tope);
END_REGION

REGION Network 24: touts topes
   RUNG wire#powerrail
      Contact( "DB902_Estado_ZonaMesa".EstadoMesas[#Mesa].Rearme_CBx )
      S_RS(operand := "DB900_Estado_Mesas".EstadoVI[#Mesa].Err_TOut_Subir_TP_E1_E3, s1 := wire#w1)
      S_Coil( "DB900_Estado_Mesas".EstadoVI[#Mesa].Error_Mx )
   END_RUNG
   RUNG wire#powerrail
      Contact( "DB1_SalidasExterioresDeMesa".Mesa[#Mesa].Subir_TP_E1E3 )
   END_RUNG wire#w1
   RUNG wire#powerrail
      Contact( "DB1_SalidasExterioresDeMesa".Mesa[#Mesa].Subir_TP_E3E1 )
   END_RUNG wire#w1
   // the same network as SCL:
   #_w1 := "DB1_SalidasExterioresDeMesa".Mesa[#Mesa].Subir_TP_E1E3 OR "DB1_SalidasExterioresDeMesa".Mesa[#Mesa].Subir_TP_E3E1;
   IF "DB902_Estado_ZonaMesa".EstadoMesas[#Mesa].Rearme_CBx THEN
       "DB900_Estado_Mesas".EstadoVI[#Mesa].Err_TOut_Subir_TP_E1_E3 := FALSE;   // RS flip-flop
   END_IF;
   IF #_w1 THEN "DB900_Estado_Mesas".EstadoVI[#Mesa].Err_TOut_Subir_TP_E1_E3 := TRUE; END_IF;
   IF "DB900_Estado_Mesas".EstadoVI[#Mesa].Err_TOut_Subir_TP_E1_E3 THEN
       "DB900_Estado_Mesas".EstadoVI[#Mesa].Error_Mx := TRUE;
   END_IF;
END_REGION

REGION Network 25: touts topes
   RUNG wire#powerrail
      Contact( "DB902_Estado_ZonaMesa".EstadoMesas[#Mesa].Rearme_CBx )
      S_RS(operand := "DB900_Estado_Mesas".EstadoVI[#Mesa].Err_TOut_Bajar_TP_E1_E3, s1 := wire#w1)
      S_Coil( "DB900_Estado_Mesas".EstadoVI[#Mesa].Error_Mx )
   END_RUNG
   RUNG wire#powerrail
      Contact( "DB1_SalidasExterioresDeMesa".Mesa[#Mesa].Bajar_TP_E1E3 )
   END_RUNG wire#w1
   RUNG wire#powerrail
      Contact( "DB1_SalidasExterioresDeMesa".Mesa[#Mesa].Bajar_TP_E3E1 )
   END_RUNG wire#w1
   // the same network as SCL:
   #_w1 := "DB1_SalidasExterioresDeMesa".Mesa[#Mesa].Bajar_TP_E1E3 OR "DB1_SalidasExterioresDeMesa".Mesa[#Mesa].Bajar_TP_E3E1;
   IF "DB902_Estado_ZonaMesa".EstadoMesas[#Mesa].Rearme_CBx THEN
       "DB900_Estado_Mesas".EstadoVI[#Mesa].Err_TOut_Bajar_TP_E1_E3 := FALSE;   // RS flip-flop
   END_IF;
   IF #_w1 THEN "DB900_Estado_Mesas".EstadoVI[#Mesa].Err_TOut_Bajar_TP_E1_E3 := TRUE; END_IF;
   IF "DB900_Estado_Mesas".EstadoVI[#Mesa].Err_TOut_Bajar_TP_E1_E3 THEN
       "DB900_Estado_Mesas".EstadoVI[#Mesa].Error_Mx := TRUE;
   END_IF;
END_REGION

REGION Network 26: TIMEOUT ATASCO
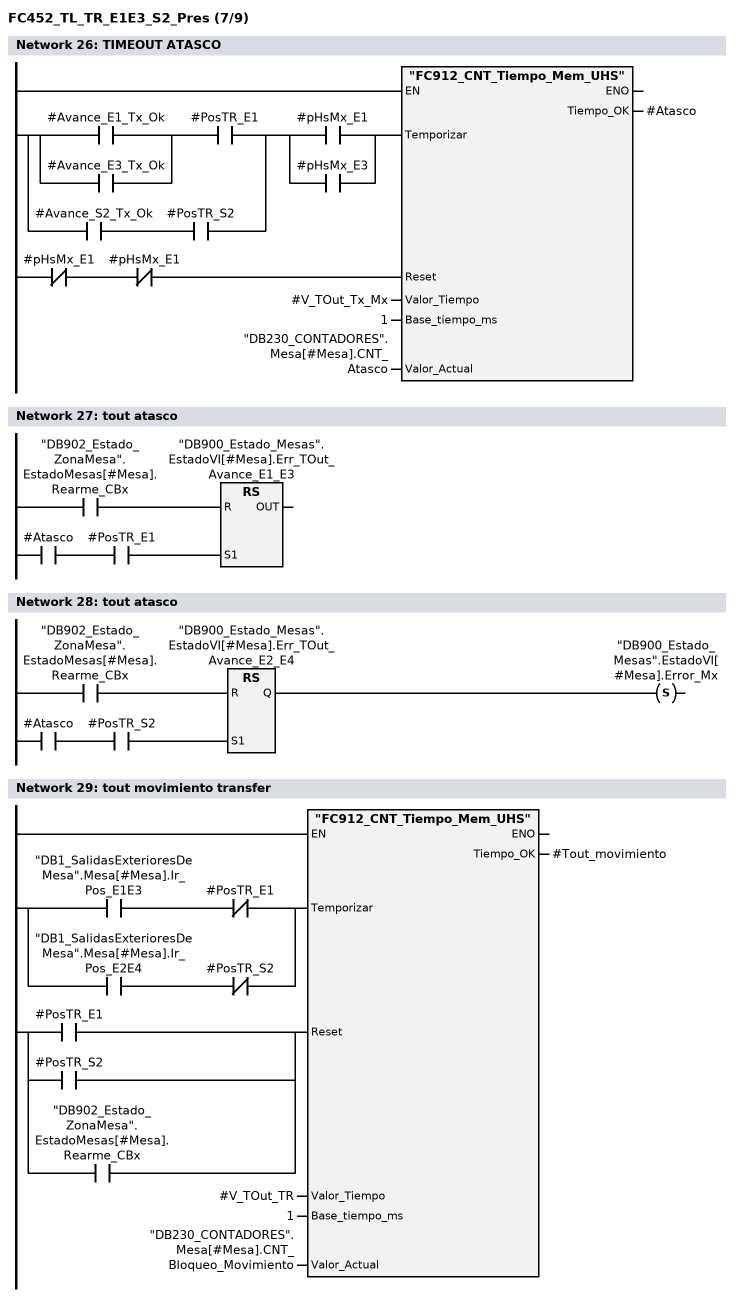
   RUNG wire#powerrail
      "FC912_CNT_Tiempo_Mem_UHS"(Temporizar := wire#w3, Reset := wire#w4, Valor_Tiempo := #V_TOut_Tx_Mx, Base_tiempo_ms := 1, Valor_Actual := "DB230_CONTADORES".Mesa[#Mesa].CNT_Atasco, Tiempo_OK => #Atasco)
   END_RUNG
   RUNG wire#powerrail
      Contact( #Avance_E1_Tx_Ok )
      wire#w1
      Contact( #PosTR_E1 )
      wire#w2
      Contact( #pHsMx_E1 )
   END_RUNG wire#w3
   RUNG wire#powerrail
      Contact( #Avance_E3_Tx_Ok )
   END_RUNG wire#w1
   RUNG wire#powerrail
      Contact( #Avance_S2_Tx_Ok )
      Contact( #PosTR_S2 )
   END_RUNG wire#w2
   RUNG wire#w2
      Contact( #pHsMx_E3 )
   END_RUNG wire#w3
   RUNG wire#powerrail
      I_Contact( #pHsMx_E1 )
      I_Contact( #pHsMx_E1 )
   END_RUNG wire#w4
   // the same network as SCL:
   "FC912_CNT_Tiempo_Mem_UHS"(Temporizar := (((#Avance_E1_Tx_Ok OR #Avance_E3_Tx_Ok) AND #PosTR_E1) OR (#Avance_S2_Tx_Ok AND #PosTR_S2)) AND (#pHsMx_E1 OR #pHsMx_E3),
                           Reset := NOT #pHsMx_E1 AND NOT #pHsMx_E1,
                           Valor_Tiempo := #V_TOut_Tx_Mx,
                           Base_tiempo_ms := 1,
                           Valor_Actual := "DB230_CONTADORES".Mesa[#Mesa].CNT_Atasco,
                           Tiempo_OK => #Atasco);
END_REGION

REGION Network 27: tout atasco
   RUNG wire#powerrail
      Contact( "DB902_Estado_ZonaMesa".EstadoMesas[#Mesa].Rearme_CBx )
      S_RS(operand := "DB900_Estado_Mesas".EstadoVI[#Mesa].Err_TOut_Avance_E1_E3, s1 := wire#w1)
   END_RUNG
   RUNG wire#powerrail
      Contact( #Atasco )
      Contact( #PosTR_E1 )
   END_RUNG wire#w1
   // the same network as SCL:
   IF "DB902_Estado_ZonaMesa".EstadoMesas[#Mesa].Rearme_CBx THEN
       "DB900_Estado_Mesas".EstadoVI[#Mesa].Err_TOut_Avance_E1_E3 := FALSE;   // RS flip-flop
   END_IF;
   IF #Atasco AND #PosTR_E1 THEN "DB900_Estado_Mesas".EstadoVI[#Mesa].Err_TOut_Avance_E1_E3 := TRUE; END_IF;
END_REGION

REGION Network 28: tout atasco
   RUNG wire#powerrail
      Contact( "DB902_Estado_ZonaMesa".EstadoMesas[#Mesa].Rearme_CBx )
      S_RS(operand := "DB900_Estado_Mesas".EstadoVI[#Mesa].Err_TOut_Avance_E2_E4, s1 := wire#w1)
      S_Coil( "DB900_Estado_Mesas".EstadoVI[#Mesa].Error_Mx )
   END_RUNG
   RUNG wire#powerrail
      Contact( #Atasco )
      Contact( #PosTR_S2 )
   END_RUNG wire#w1
   // the same network as SCL:
   IF "DB902_Estado_ZonaMesa".EstadoMesas[#Mesa].Rearme_CBx THEN
       "DB900_Estado_Mesas".EstadoVI[#Mesa].Err_TOut_Avance_E2_E4 := FALSE;   // RS flip-flop
   END_IF;
   IF #Atasco AND #PosTR_S2 THEN "DB900_Estado_Mesas".EstadoVI[#Mesa].Err_TOut_Avance_E2_E4 := TRUE; END_IF;
   IF "DB900_Estado_Mesas".EstadoVI[#Mesa].Err_TOut_Avance_E2_E4 THEN
       "DB900_Estado_Mesas".EstadoVI[#Mesa].Error_Mx := TRUE;
   END_IF;
END_REGION

REGION Network 29: tout movimiento transfer
   RUNG wire#powerrail
      "FC912_CNT_Tiempo_Mem_UHS"(Temporizar := wire#w1, Reset := wire#w2, Valor_Tiempo := #V_TOut_TR, Base_tiempo_ms := 1, Valor_Actual := "DB230_CONTADORES".Mesa[#Mesa].CNT_Bloqueo_Movimiento, Tiempo_OK => #Tout_movimiento)
   END_RUNG
   RUNG wire#powerrail
      Contact( "DB1_SalidasExterioresDeMesa".Mesa[#Mesa].Ir_Pos_E1E3 )
      I_Contact( #PosTR_E1 )
   END_RUNG wire#w1
   RUNG wire#powerrail
      Contact( "DB1_SalidasExterioresDeMesa".Mesa[#Mesa].Ir_Pos_E2E4 )
      I_Contact( #PosTR_S2 )
   END_RUNG wire#w1
   RUNG wire#powerrail
      Contact( #PosTR_E1 )
   END_RUNG wire#w2
   RUNG wire#powerrail
      Contact( #PosTR_S2 )
   END_RUNG wire#w2
   RUNG wire#powerrail
      Contact( "DB902_Estado_ZonaMesa".EstadoMesas[#Mesa].Rearme_CBx )
   END_RUNG wire#w2
   // the same network as SCL:
   "FC912_CNT_Tiempo_Mem_UHS"(Temporizar := ("DB1_SalidasExterioresDeMesa".Mesa[#Mesa].Ir_Pos_E1E3 AND NOT #PosTR_E1) OR ("DB1_SalidasExterioresDeMesa".Mesa[#Mesa].Ir_Pos_E2E4 AND NOT #PosTR_S2),
                           Reset := #PosTR_E1 OR #PosTR_S2 OR "DB902_Estado_ZonaMesa".EstadoMesas[#Mesa].Rearme_CBx,
                           Valor_Tiempo := #V_TOut_TR,
                           Base_tiempo_ms := 1,
                           Valor_Actual := "DB230_CONTADORES".Mesa[#Mesa].CNT_Bloqueo_Movimiento,
                           Tiempo_OK => #Tout_movimiento);
END_REGION

REGION Network 30: tout
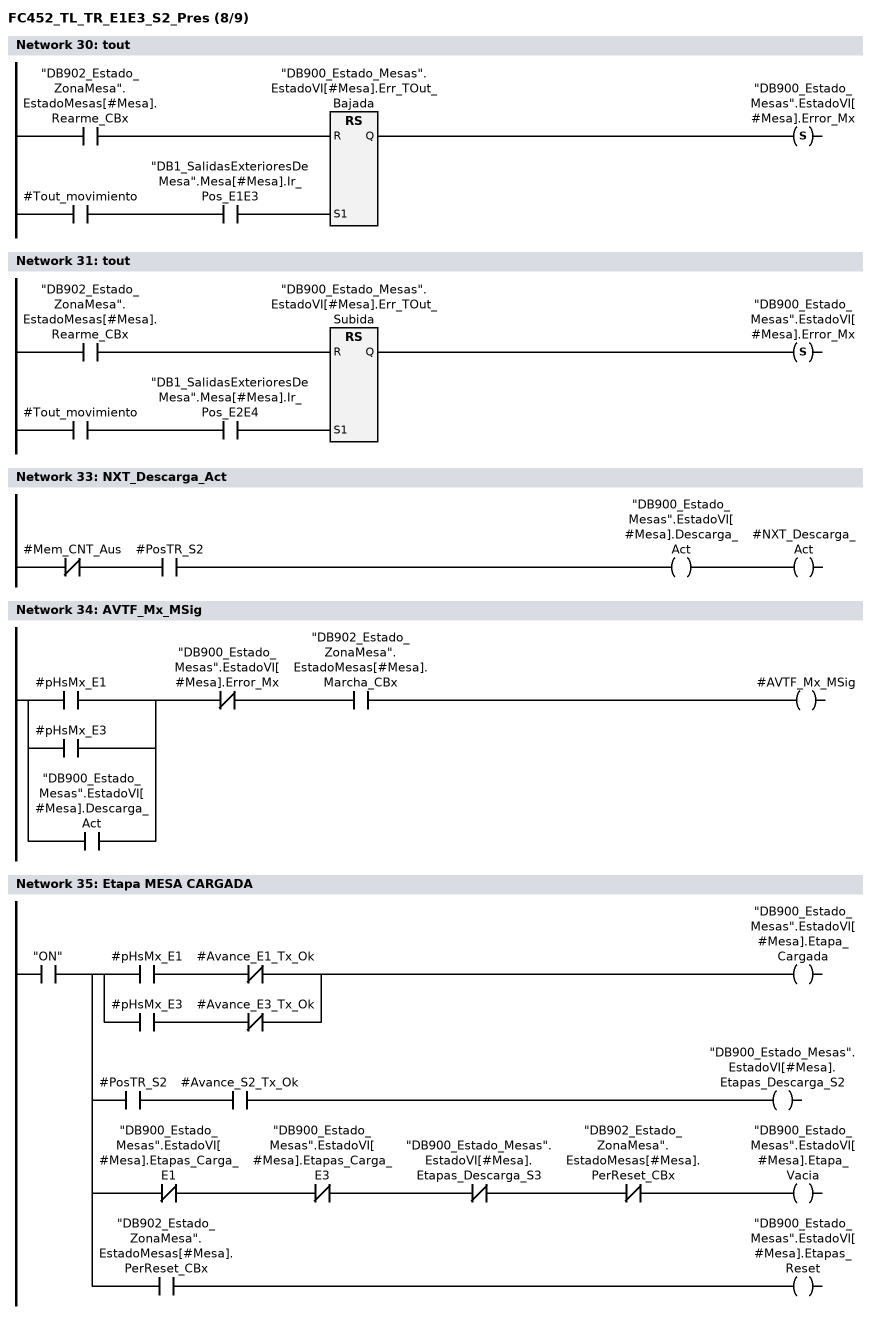
   RUNG wire#powerrail
      Contact( "DB902_Estado_ZonaMesa".EstadoMesas[#Mesa].Rearme_CBx )
      S_RS(operand := "DB900_Estado_Mesas".EstadoVI[#Mesa].Err_TOut_Bajada, s1 := wire#w1)
      S_Coil( "DB900_Estado_Mesas".EstadoVI[#Mesa].Error_Mx )
   END_RUNG
   RUNG wire#powerrail
      Contact( #Tout_movimiento )
      Contact( "DB1_SalidasExterioresDeMesa".Mesa[#Mesa].Ir_Pos_E1E3 )
   END_RUNG wire#w1
   // the same network as SCL:
   #_w1 := #Tout_movimiento AND "DB1_SalidasExterioresDeMesa".Mesa[#Mesa].Ir_Pos_E1E3;
   IF "DB902_Estado_ZonaMesa".EstadoMesas[#Mesa].Rearme_CBx THEN
       "DB900_Estado_Mesas".EstadoVI[#Mesa].Err_TOut_Bajada := FALSE;   // RS flip-flop
   END_IF;
   IF #_w1 THEN "DB900_Estado_Mesas".EstadoVI[#Mesa].Err_TOut_Bajada := TRUE; END_IF;
   IF "DB900_Estado_Mesas".EstadoVI[#Mesa].Err_TOut_Bajada THEN
       "DB900_Estado_Mesas".EstadoVI[#Mesa].Error_Mx := TRUE;
   END_IF;
END_REGION

REGION Network 31: tout
   RUNG wire#powerrail
      Contact( "DB902_Estado_ZonaMesa".EstadoMesas[#Mesa].Rearme_CBx )
      S_RS(operand := "DB900_Estado_Mesas".EstadoVI[#Mesa].Err_TOut_Subida, s1 := wire#w1)
      S_Coil( "DB900_Estado_Mesas".EstadoVI[#Mesa].Error_Mx )
   END_RUNG
   RUNG wire#powerrail
      Contact( #Tout_movimiento )
      Contact( "DB1_SalidasExterioresDeMesa".Mesa[#Mesa].Ir_Pos_E2E4 )
   END_RUNG wire#w1
   // the same network as SCL:
   #_w1 := #Tout_movimiento AND "DB1_SalidasExterioresDeMesa".Mesa[#Mesa].Ir_Pos_E2E4;
   IF "DB902_Estado_ZonaMesa".EstadoMesas[#Mesa].Rearme_CBx THEN
       "DB900_Estado_Mesas".EstadoVI[#Mesa].Err_TOut_Subida := FALSE;   // RS flip-flop
   END_IF;
   IF #_w1 THEN "DB900_Estado_Mesas".EstadoVI[#Mesa].Err_TOut_Subida := TRUE; END_IF;
   IF "DB900_Estado_Mesas".EstadoVI[#Mesa].Err_TOut_Subida THEN
       "DB900_Estado_Mesas".EstadoVI[#Mesa].Error_Mx := TRUE;
   END_IF;
END_REGION

REGION Network 33: NXT_Descarga_Act
   RUNG wire#powerrail
      I_Contact( #Mem_CNT_Aus )
      Contact( #PosTR_S2 )
      Coil( "DB900_Estado_Mesas".EstadoVI[#Mesa].Descarga_Act )
      Coil( #NXT_Descarga_Act )
   END_RUNG
   // the same network as SCL:
   "DB900_Estado_Mesas".EstadoVI[#Mesa].Descarga_Act := NOT #Mem_CNT_Aus AND #PosTR_S2;
   #NXT_Descarga_Act := NOT #Mem_CNT_Aus AND #PosTR_S2;
END_REGION

REGION Network 34: AVTF_Mx_MSig
   RUNG wire#powerrail
      Contact( #pHsMx_E1 )
      wire#w1
      I_Contact( "DB900_Estado_Mesas".EstadoVI[#Mesa].Error_Mx )
      Contact( "DB902_Estado_ZonaMesa".EstadoMesas[#Mesa].Marcha_CBx )
      Coil( #AVTF_Mx_MSig )
   END_RUNG
   RUNG wire#powerrail
      Contact( #pHsMx_E3 )
   END_RUNG wire#w1
   RUNG wire#powerrail
      Contact( "DB900_Estado_Mesas".EstadoVI[#Mesa].Descarga_Act )
   END_RUNG wire#w1
   // the same network as SCL:
   #AVTF_Mx_MSig := (#pHsMx_E1 OR #pHsMx_E3 OR "DB900_Estado_Mesas".EstadoVI[#Mesa].Descarga_Act) AND NOT "DB900_Estado_Mesas".EstadoVI[#Mesa].Error_Mx AND "DB902_Estado_ZonaMesa".EstadoMesas[#Mesa].Marcha_CBx;
END_REGION

REGION Network 35: Etapa MESA CARGADA
   RUNG wire#powerrail
      Contact( "ON" )
      wire#w1
      Contact( #pHsMx_E1 )
      I_Contact( #Avance_E1_Tx_Ok )
      wire#w2
      Coil( "DB900_Estado_Mesas".EstadoVI[#Mesa].Etapa_Cargada )
   END_RUNG
   RUNG wire#w1
      Contact( #pHsMx_E3 )
      I_Contact( #Avance_E3_Tx_Ok )
   END_RUNG wire#w2
   RUNG wire#w1
      Contact( #PosTR_S2 )
      Contact( #Avance_S2_Tx_Ok )
      Coil( "DB900_Estado_Mesas".EstadoVI[#Mesa].Etapas_Descarga_S2 )
   END_RUNG
   RUNG wire#w1
      I_Contact( "DB900_Estado_Mesas".EstadoVI[#Mesa].Etapas_Carga_E1 )
      I_Contact( "DB900_Estado_Mesas".EstadoVI[#Mesa].Etapas_Carga_E3 )
      I_Contact( "DB900_Estado_Mesas".EstadoVI[#Mesa].Etapas_Descarga_S3 )
      I_Contact( "DB902_Estado_ZonaMesa".EstadoMesas[#Mesa].PerReset_CBx )
      Coil( "DB900_Estado_Mesas".EstadoVI[#Mesa].Etapa_Vacia )
   END_RUNG
   RUNG wire#w1
      Contact( "DB902_Estado_ZonaMesa".EstadoMesas[#Mesa].PerReset_CBx )
      Coil( "DB900_Estado_Mesas".EstadoVI[#Mesa].Etapas_Reset )
   END_RUNG
   // the same network as SCL:
   "DB900_Estado_Mesas".EstadoVI[#Mesa].Etapa_Cargada := "ON" AND ((#pHsMx_E1 AND NOT #Avance_E1_Tx_Ok) OR (#pHsMx_E3 AND NOT #Avance_E3_Tx_Ok));
   "DB900_Estado_Mesas".EstadoVI[#Mesa].Etapas_Descarga_S2 := "ON" AND #PosTR_S2 AND #Avance_S2_Tx_Ok;
   "DB900_Estado_Mesas".EstadoVI[#Mesa].Etapa_Vacia := "ON" AND NOT "DB900_Estado_Mesas".EstadoVI[#Mesa].Etapas_Carga_E1 AND NOT "DB900_Estado_Mesas".EstadoVI[#Mesa].Etapas_Carga_E3 AND NOT "DB900_Estado_Mesas".EstadoVI[#Mesa].Etapas_Descarga_S3 AND NOT "DB902_Estado_ZonaMesa".EstadoMesas[#Mesa].PerReset_CBx;
   "DB900_Estado_Mesas".EstadoVI[#Mesa].Etapas_Reset := "ON" AND "DB902_Estado_ZonaMesa".EstadoMesas[#Mesa].PerReset_CBx;
END_REGION

REGION Network 36: Entradas Mesas
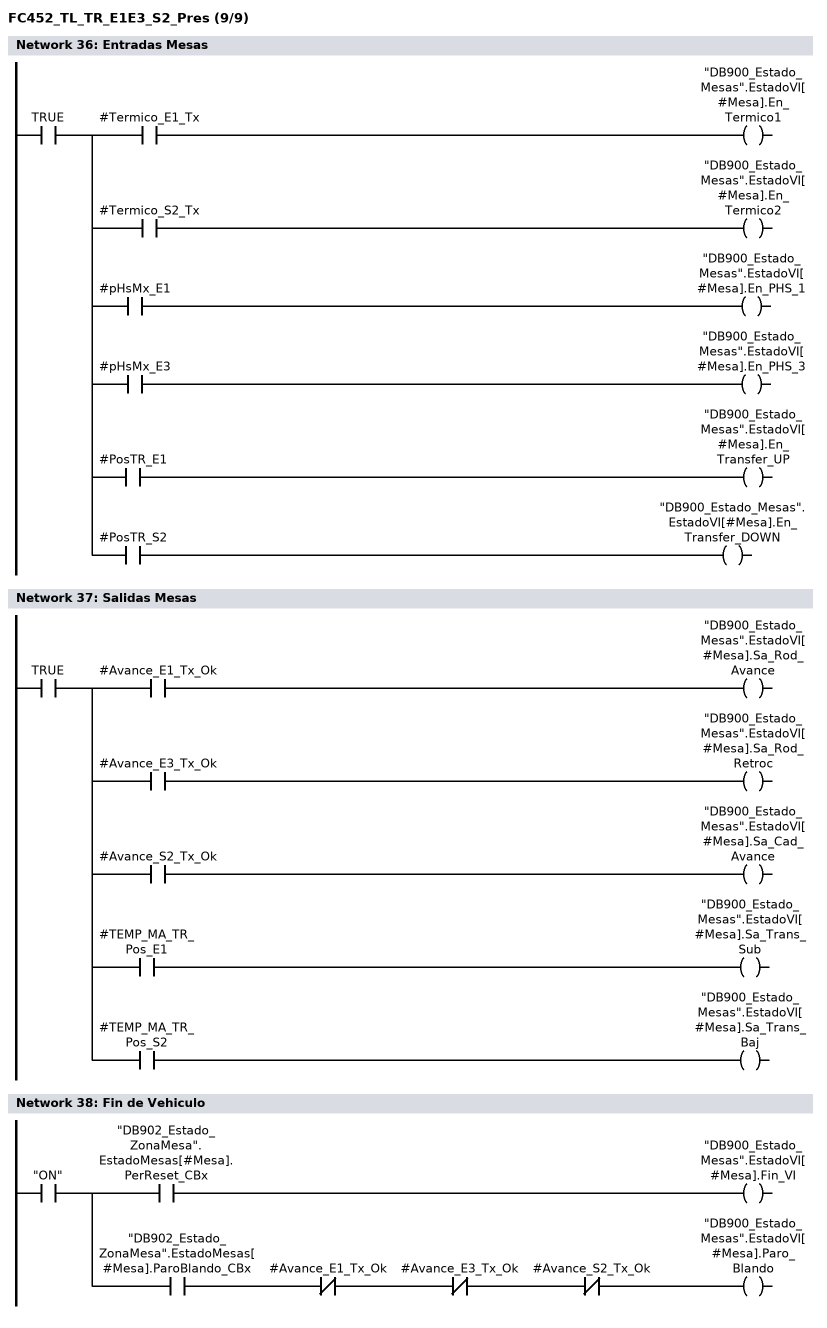
   RUNG wire#powerrail
      Contact( TRUE )
      wire#w1
      Contact( #Termico_E1_Tx )
      Coil( "DB900_Estado_Mesas".EstadoVI[#Mesa].En_Termico1 )
   END_RUNG
   RUNG wire#w1
      Contact( #Termico_S2_Tx )
      Coil( "DB900_Estado_Mesas".EstadoVI[#Mesa].En_Termico2 )
   END_RUNG
   RUNG wire#w1
      Contact( #pHsMx_E1 )
      Coil( "DB900_Estado_Mesas".EstadoVI[#Mesa].En_PHS_1 )
   END_RUNG
   RUNG wire#w1
      Contact( #pHsMx_E3 )
      Coil( "DB900_Estado_Mesas".EstadoVI[#Mesa].En_PHS_3 )
   END_RUNG
   RUNG wire#w1
      Contact( #PosTR_E1 )
      Coil( "DB900_Estado_Mesas".EstadoVI[#Mesa].En_Transfer_UP )
   END_RUNG
   RUNG wire#w1
      Contact( #PosTR_S2 )
      Coil( "DB900_Estado_Mesas".EstadoVI[#Mesa].En_Transfer_DOWN )
   END_RUNG
   // the same network as SCL:
   "DB900_Estado_Mesas".EstadoVI[#Mesa].En_Termico1 := TRUE AND #Termico_E1_Tx;
   "DB900_Estado_Mesas".EstadoVI[#Mesa].En_Termico2 := TRUE AND #Termico_S2_Tx;
   "DB900_Estado_Mesas".EstadoVI[#Mesa].En_PHS_1 := TRUE AND #pHsMx_E1;
   "DB900_Estado_Mesas".EstadoVI[#Mesa].En_PHS_3 := TRUE AND #pHsMx_E3;
   "DB900_Estado_Mesas".EstadoVI[#Mesa].En_Transfer_UP := TRUE AND #PosTR_E1;
   "DB900_Estado_Mesas".EstadoVI[#Mesa].En_Transfer_DOWN := TRUE AND #PosTR_S2;
END_REGION

REGION Network 37: Salidas Mesas
   RUNG wire#powerrail
      Contact( TRUE )
      wire#w1
      Contact( #Avance_E1_Tx_Ok )
      Coil( "DB900_Estado_Mesas".EstadoVI[#Mesa].Sa_Rod_Avance )
   END_RUNG
   RUNG wire#w1
      Contact( #Avance_E3_Tx_Ok )
      Coil( "DB900_Estado_Mesas".EstadoVI[#Mesa].Sa_Rod_Retroc )
   END_RUNG
   RUNG wire#w1
      Contact( #Avance_S2_Tx_Ok )
      Coil( "DB900_Estado_Mesas".EstadoVI[#Mesa].Sa_Cad_Avance )
   END_RUNG
   RUNG wire#w1
      Contact( #TEMP_MA_TR_Pos_E1 )
      Coil( "DB900_Estado_Mesas".EstadoVI[#Mesa].Sa_Trans_Sub )
   END_RUNG
   RUNG wire#w1
      Contact( #TEMP_MA_TR_Pos_S2 )
      Coil( "DB900_Estado_Mesas".EstadoVI[#Mesa].Sa_Trans_Baj )
   END_RUNG
   // the same network as SCL:
   "DB900_Estado_Mesas".EstadoVI[#Mesa].Sa_Rod_Avance := TRUE AND #Avance_E1_Tx_Ok;
   "DB900_Estado_Mesas".EstadoVI[#Mesa].Sa_Rod_Retroc := TRUE AND #Avance_E3_Tx_Ok;
   "DB900_Estado_Mesas".EstadoVI[#Mesa].Sa_Cad_Avance := TRUE AND #Avance_S2_Tx_Ok;
   "DB900_Estado_Mesas".EstadoVI[#Mesa].Sa_Trans_Sub := TRUE AND #TEMP_MA_TR_Pos_E1;
   "DB900_Estado_Mesas".EstadoVI[#Mesa].Sa_Trans_Baj := TRUE AND #TEMP_MA_TR_Pos_S2;
END_REGION

REGION Network 38: Fin de Vehiculo
   RUNG wire#powerrail
      Contact( "ON" )
      wire#w1
      Contact( "DB902_Estado_ZonaMesa".EstadoMesas[#Mesa].PerReset_CBx )
      Coil( "DB900_Estado_Mesas".EstadoVI[#Mesa].Fin_VI )
   END_RUNG
   RUNG wire#w1
      Contact( "DB902_Estado_ZonaMesa".EstadoMesas[#Mesa].ParoBlando_CBx )
      I_Contact( #Avance_E1_Tx_Ok )
      I_Contact( #Avance_E3_Tx_Ok )
      I_Contact( #Avance_S2_Tx_Ok )
      Coil( "DB900_Estado_Mesas".EstadoVI[#Mesa].Paro_Blando )
   END_RUNG
   // the same network as SCL:
   "DB900_Estado_Mesas".EstadoVI[#Mesa].Fin_VI := "ON" AND "DB902_Estado_ZonaMesa".EstadoMesas[#Mesa].PerReset_CBx;
   "DB900_Estado_Mesas".EstadoVI[#Mesa].Paro_Blando := "ON" AND "DB902_Estado_ZonaMesa".EstadoMesas[#Mesa].ParoBlando_CBx AND NOT #Avance_E1_Tx_Ok AND NOT #Avance_E3_Tx_Ok AND NOT #Avance_S2_Tx_Ok;
END_REGION
END_FUNCTION
